INTERFACE I_DrawableShape EXTENDS I_Disposable

METHOD Clone : I_DrawableShape
VAR_INPUT
END_VAR
END_METHOD

METHOD Draw
VAR_INPUT
END_VAR
END_METHOD

END_INTERFACE

(* stored: Version 1.1.0.1, ProductVersion 3.1.4024.12
   Itf I_DrawableShape: Id {845d4f0e-7686-422c-bfa9-9f7d44dcc274}
   Method Clone: Id {267796f6-e282-4810-b929-b9e4e73721a4}
   Method Draw: Id {5fc940af-ada7-4e36-a96a-1e791eebb941} *)
